Universal Robots URScript: straight floor demo.script

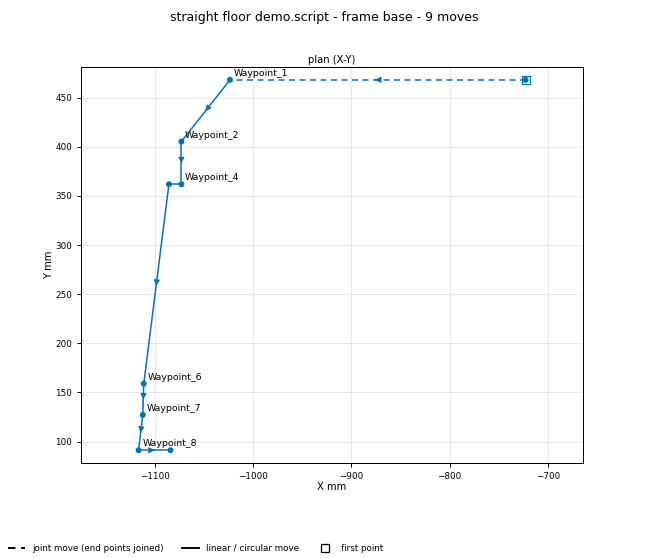
[picture p0: tool path of straight floor demo.script in frame base, 9 of 9 moves have a stored position in this frame; points joined in program order, loops and branches not executed]
def straight_floor_demo():
  global _hidden_verificationVariable=0
  set_target_payload(10.800000, [-0.001000, -0.053000, 0.068000], [0.081228, 0.081228, 0.081228, 0.000000, 0.000000, 0.000000])
  set_gravity([0.0, 0.0, 9.82])
  set_standard_analog_input_domain(0, 1)
  set_standard_analog_input_domain(1, 1)
  set_tool_analog_input_domain(0, 1)
  set_tool_analog_input_domain(1, 1)
  set_analog_outputdomain(0, 0)
  set_analog_outputdomain(1, 0)
  set_input_actions_to_default()
  set_safety_mode_transition_hardness(1)
  set_tcp(p[-0.0095,-0.328,0.10573,1.2092,-1.2092,1.2092])
  set_tool_communication(False, 115200, 0, 1, 1.5, 3.5)
  set_tool_output_mode(0)
  set_tool_digital_output_mode(0, 1)
  set_tool_digital_output_mode(1, 1)
  set_tool_voltage(0)
  global robot_number=2
  global Point_1=p[0.0,0.0,0.0,0.0,0.0,0.0]
  global Point_2=p[0.0,0.0,0.0,0.0,0.0,0.0]
  # begin: URCap Installation Node
  #   Source: UR Connect, 1.13.79, Universal Robots
  #   Type: UR Connect
  myurRPC = rpc_factory("xmlrpc","http://127.0.0.1:40474")
  # end: URCap Installation Node
  # begin: URCap Installation Node
  #   Source: MachineLogic for Universal Robots, 3.1.7, Vention Inc.
  #   Type: MachineLogic for Universal Robots
  def waitForResponse(expected_response_vention, cname_vention):
  response_vention = socket_read_string(cname_vention,timeout=15)
  while response_vention != expected_response_vention:
  sleep(0.01)
  response_vention = socket_read_string(cname_vention,timeout=15)
  end
  sleep(0.01)
  sync()
  end
  def sendString(string_vention, expected_response_vention, cname_vention):
  socket_send_string(str_cat(string_vention,";"), cname_vention)
  response_vention = socket_read_string(cname_vention,timeout=15)
  if(response_vention == "nAck"):
  popup("nAck received")
  end
  while response_vention != expected_response_vention:
  sleep(0.01)
  response_vention = socket_read_string(cname_vention,timeout=15)
  if(response_vention == "nAck"):
  popup("nAck received")
  end
  end
  sleep(0.01)
  sync()
  end
  def sendStringNAck(string_vention, expected_response_vention, cname_vention):
  socket_send_string(str_cat(string_vention,";"), cname_vention)
  response_vention = socket_read_string(cname_vention,timeout=15)
  if(response_vention == "nAck"):
  popup("nAck received")
  end
  while(response_vention != expected_response_vention and response_vention != "nAck"):
  sleep(0.01)
  response_vention = socket_read_string(cname_vention,timeout=15)
  if(response_vention == "nAck"):
  popup("nAck received",blocking=True)
  end
  end
  sleep(0.01)
  sync()
  end
  def sendStringWithTimeout(string_vention, expected_response_vention, cname_vention):
  socket_send_string(str_cat(string_vention,";"), cname_vention)
  response_vention = socket_read_string(cname_vention,timeout=10)
  if(response_vention == "nAck"):
  popup("nAck received"+string_vention)
  end
  sleep(0.01)
  sync()
  end
  def pollString(string_vention, expected_response_vention, cname_vention):
  socket_send_string(str_cat(string_vention,";"), cname_vention)
  response_vention = socket_read_string(cname_vention,timeout=15)
  if(response_vention == "nAck"):
  popup("nAck received")
  end
  while response_vention != expected_response_vention:
  sleep(1)
  socket_send_string(str_cat(string_vention,";"), cname_vention)
  response_vention = socket_read_string(cname_vention,timeout=15)
  if(response_vention == "nAck"):
  popup("nAck received")
  end
  end
  sleep(0.01)
  sync()
  end
  def sendVariable(var_vention, data_vention, expected_response_vention, cname_vention):
  socket_set_var(var_vention, data_vention, cname_vention)
  response_vention = socket_read_string(cname_vention,timeout=15)
  if(response_vention == "nAck"):
  popup("nAck received")
  end
  while response_vention != expected_response_vention:
  sleep(0.01)
  response_vention = socket_read_string(cname_vention,timeout=15)
  if(response_vention == "nAck"):
  popup("nAck received")
  end
  end
  sleep(0.01)
  sync()
  end
  def intToString(integer_vention,cname_vention):
  stringFix=""
  multiplier_vention123=1
  if integer_vention<0:
  stringFix="-"
  multiplier_vention123=-1
  end
  socket_set_var("GetString",integer_vention*multiplier_vention123,cname_vention)
  string_vention=""
  while string_vention=="":
  sleep(0.01)
  string_vention=socket_read_string(cname_vention,timeout=15)
  end
  sleep(0.01)
  sync()
  string_vention=stringFix+string_vention
  return string_vention
  end
  string_vention=""
  isVentionMovementBusy = False
  isVentionParallelMovementSendingScript = False
  ventionThreadHandle = 1
  isVentionMovementBusyMachineMotion1 = False
  isVentionParallelMovementSendingScriptMachineMotion1 = False
  socket_vention = socket_open("192.168.3.52", 9999, "MachineMotion1")
  if socket_vention==False:
  popup("Check configuration, can't connect to MachineMotion")
  end
  waitForResponse("MachineMotion connection established", "MachineMotion1")
  sendString("isReady", "MachineMotion isReady = true", "MachineMotion1")
  sendStringWithTimeout("setURCapVersion2", "setURCapVersion loaded", "MachineMotion1")
  sendString("SET speed_v2 1000000", "Ack", "MachineMotion1")
  sendString("SET acceleration_v2 100000", "Ack", "MachineMotion1")
  sendString("SET de_axis_1_microsteps_config 8", "Ack", "MachineMotion1")
  sendString("SET de_axis_1_mechanical_gain_config_v2 150000.0", "Ack", "MachineMotion1")
  sendString("SET de_axis_1_direction_config 1", "Ack", "MachineMotion1")
  sendString("SET de_axis_1_type_config Custom Actuator ", "Ack", "MachineMotion1")
  sendString("de_axis_1_config_exec", "Ack", "MachineMotion1")
  # end: URCap Installation Node
  # begin: URCap Installation Node
  #   Source: WireTank Serial, 4.9.0, WireTank, LLC
  #   Type: WireTank Serial
  WTSerialBridge = rpc_factory("xmlrpc","http://127.0.0.1:40511/RPC2")
  # end: URCap Installation Node
  step_count_cfc27bff_3819_45be_bfcf_d52b1b1e9d2e = 0.0
  thread Step_Counter_Thread_60c3a4a9_e978_4eed_be39_a7f2d0dbddbc():
    while (True):
      step_count_cfc27bff_3819_45be_bfcf_d52b1b1e9d2e = step_count_cfc27bff_3819_45be_bfcf_d52b1b1e9d2e + 1.0
      sync()
    end
  end
  run Step_Counter_Thread_60c3a4a9_e978_4eed_be39_a7f2d0dbddbc()
  global Waypoint_3_p=p[-.722693512961, .468114258570, -.058678755751, -2.111593641716, .331077455790, 2.041155761858]
  global Waypoint_3_q=[-1.117944307747626, -0.9479933470459523, 2.696181567308242, -3.27753173466739, -1.5847299872922047, 5.455842043959539]
  global Waypoint_1_p=p[-1.023508508072, .468114258579, -.058678755757, -2.111593641715, .331077455789, 2.041155761858]
  global Waypoint_1_q=[-0.7503212133990687, -0.9486703437617798, 2.3420866171466272, -2.9208342037596644, -1.5690940062152308, 5.8232421875]
  global Waypoint_2_p=p[-1.072965120894, .405321236272, -.050994421483, 2.238822905034, .005513598899, -2.156859240811]
  global Waypoint_2_q=[-0.7493843284088637, -0.9418009390670319, 2.2640598169838597, -2.8509786388692766, -1.582374607975213, 5.508504185773622]
  global Waypoint_4_p=p[-1.072965120840, .361906241167, -.050994421477, 2.238822905035, .005513598898, -2.156859240810]
  global Waypoint_4_q=[-0.7105926135525156, -0.9494985814034127, 2.2940700773317158, -2.8729054351797316, -1.5807736117674498, 5.547260315541911]
  global Waypoint_5_p=p[-1.085671078638, .361906241000, -.050994421407, -2.207475107603, .158359319102, 2.130004340164]
  global Waypoint_5_q=[-0.6561308013785698, -0.9528004094341185, 2.306717754213087, -2.8812627354432063, -1.5722086160524071, 5.749692039586737]
  global Waypoint_6_p=p[-1.111256290834, .158940108024, -.050994421193, -2.207475107614, .158359319108, 2.130004340158]
  global Waypoint_6_q=[-0.420521134668129, -0.9636000838567087, 2.3561240401381305, -2.920910067371023, -1.5622556429313512, 5.985078478804208]
  global Waypoint_7_p=p[-1.112304890464, .127175725525, -.050994421004, 2.250573753646, -.021660072920, -2.168735455876]
  global Waypoint_7_q=[-0.4292241528726244, -0.9632624599277371, 2.3534346923792087, -2.9176831611850744, -1.5678386625550331, 5.8525134307567335]
  global Waypoint_8_p=p[-1.116577638718, .091212938315, -.050994420874, 2.250573753649, -.021660072923, -2.168735455870]
  global Waypoint_8_q=[-0.38475971841863643, -0.9636162631979861, 2.3553828562352095, -2.9194882006238942, -1.5659556053016495, 5.8969364506940165]
  global Waypoint_9_p=p[-1.084025351057, .091212938245, -.050994420812, 2.250573753650, -.021660072923, -2.168735455869]
  global Waypoint_9_q=[-0.4010592963416233, -0.9725723650263625, 2.401883630590324, -2.956945909577499, -1.56665932156098, 5.880644499352385]
  while (True):
    $ 2 "Robot Program"
    $ 3 "Folder1"
    $ 6 "MoveJ"
    $ 7 "Waypoint_3" "breakAfter"
    movej(get_inverse_kin(Waypoint_3_p, qnear=Waypoint_3_q), a=1.3962634015954636, v=1.0471975511965976)
    $ 8 "Waypoint_1" "breakAfter"
    movej(get_inverse_kin(Waypoint_1_p, qnear=Waypoint_1_q), a=1.3962634015954636, v=1.0471975511965976)
    $ 9 "MoveL"
    $ 10 "Waypoint_2" "breakAfter"
    movel(Waypoint_2_p, a=1.2, v=0.02)
    $ 11 "Waypoint_4" "breakAfter"
    movel(Waypoint_4_p, a=1.2, v=0.02)
    $ 12 "Waypoint_5" "breakAfter"
    movel(Waypoint_5_p, a=1.2, v=0.02)
    $ 13 "Waypoint_6" "breakAfter"
    movel(Waypoint_6_p, a=1.2, v=0.02)
    $ 14 "Waypoint_7" "breakAfter"
    movel(Waypoint_7_p, a=1.2, v=0.02)
    $ 15 "Waypoint_8" "breakAfter"
    movel(Waypoint_8_p, a=1.2, v=0.02)
    $ 16 "Waypoint_9" "breakAfter"
    movel(Waypoint_9_p, a=1.2, v=0.02)
  end
end
